{attribute 'qualified_only'}
{attribute 'strict'}
TYPE E_DB_QUERY_STATE :
(
	IDLE_STATE,
    ERROR_STATE,
    SELECT_POST_LAST_RUN,
    SELECT_POST_LAST_RUN_ID,
    SELECT_VD_BY_NO,
    INSERT_RUN,
    INSERT_RUN_VD,
    SELECT_LAST_CALIBRATION_ID,
    INSERT_CALIBRATION,
    INSERT_CALIBRATION_VALUES,
    SELECT_ALL_SYSTEM,
    SELECT_LAST_SYSTEM_ID,
    INSERT_SYS_PARAMETERS,
    SELECT_ALL_METHODS,
    SELECT_WHOLE_METHODS,
    SELECT_ALL_ACTV_METHODS,
    INSERT_NEW_METHOD,
    UPDATE_DEACTV_METHOD,
    SELECT_VOLUME_DATA,
    INSERT_VOLUME_DATA,
    INSERT_USER,
    SELECT_ALL_USERS,
    SELECT_ALL_CURRENT_USERS
);
END_TYPE

(* stored: Version 1.1.0.1, ProductVersion 3.1.4024.15
   DUT E_DB_QUERY_STATE: Id {1492bc47-394d-4d44-a5ab-b3db879d10f1} *)
